INTERFACE I_SystemCalibration


METHOD IsCalibrated : BOOL
END_METHOD

END_INTERFACE

(* stored: Version 1.1.0.1
   Itf I_SystemCalibration: Id {48301cdf-562c-4c97-ba90-6ac51224f9e7}
   Method IsCalibrated: Id {1b048ef3-40fe-4063-b477-6ec0325a4c86} *)
